// TwinCAT 3 PLC project Untitled1
// ProgramVersion: 3.1.4023.0
// libraries:
//   Tc2_MC2, * (Beckhoff Automation GmbH)
//   Tc2_Standard, * (Beckhoff Automation GmbH)
//   Tc2_System, * (Beckhoff Automation GmbH)
//   Tc3_Module, * (Beckhoff Automation GmbH)
// project tree:
//   DUTs/ stAxisIN.TcDUT, stAxisInterface.TcDUT, stAxisOut.TcDUT
//   GVLs/ GVL_Axis.TcGVL
//   / PlcTask.TcTTO
//   POUs/ FB_Motion.TcPOU, MAIN.TcPOU
// real-time tasks:
//   TASK PlcTask: cycle T#10ms, priority 20, ADS port 350
// motion (NC):
//   TASK NC-Task 1 SAF: cycle T#2ms, priority 4, ADS port 501
//   TASK NC-Task 1 SVB: cycle T#10ms, priority 8, ADS port 511
//   AXIS Axis 1 (id 1)
//     OtherSettings: AllowMotionCmdToSlave=true
//     encoder EncType=1
//     drive DrvType=5
//       Analog: TorqueSetpointScale=10, ScaleFactorActTorque=0.1
//       TimeComp: TaskDelayCycles=1
//     controller CtrType=1
//       CtrPara: PriorControlFactor=1
//         Observer: BandWidth=20
// variable links:
//   Untitled1/Untitled1 Instance <-> NC-Task 1 SAF/Axes/Axis 1
//     PlcTask Inputs/GVL_Axis.Axis1.NcToPlc <-> Outputs/ToPlc
//     PlcTask Outputs/GVL_Axis.Axis1.PlcToNc <-> Inputs/FromPlc

CONFIGURATION Untitled1
    RESOURCE PLC ON TwinCAT3
        TASK PlcTask(INTERVAL := T#10ms, PRIORITY := 20);
        PROGRAM MAIN WITH PlcTask : MAIN;
    END_RESOURCE
END_CONFIGURATION

// ---- DUTs/stAxisIN.TcDUT
TYPE stAxisIN :
STRUCT

bPower	 :	BOOL;
bStop	:	BOOL;
bMoveAbs	:	BOOL;
bReset	:	bOOL;

fOverride	:	LREAL;
fPosition	:	LREAL;
fVelocity	:	LREAL;


END_STRUCT
END_TYPE

// ---- DUTs/stAxisInterface.TcDUT
TYPE stAxisInterface :
STRUCT
	

IN	:	stAxisIN;
OUT	:	stAxisOUT;


END_STRUCT
END_TYPE

// ---- DUTs/stAxisOut.TcDUT
TYPE stAxisOut :
STRUCT
	
bPowerErr	:	BOOL;
bPowerEnabled	:	BOOL;
bPowerACTIVE	:	BOOL;

bStopDone	:	BOOL;
bStopActive	:	BOOL;
bStopErr	:	BOOL;

bMoveAbsDone	:	BOOL;
bMoveAbsBusy	:	BOOL;
bMoveAbsActive	:	BOOL;
bMoveAbsErr		:	BOOL;

bResetDone	:	BOOL;
bResetErr	:	BOOL;	

END_STRUCT
END_TYPE

// ---- GVLs/GVL_Axis.TcGVL
VAR_GLOBAL
	
Axis1 : AXIS_REF;
stAxis1	:	stAxisInterface;


END_VAR

// ---- POUs/MAIN.TcPOU
PROGRAM MAIN
VAR
	nState: INT;
	bButton	:	BOOL;
	fbMotion	:	FB_Motion;
	T1: TON;
END_VAR



stAxis1.IN.bPower	:=	TRUE;
stAxis1.IN.fOverride	:=	100;

fbMotion(Axis:=Axis1 , staxisinterface:=stAxis1 );
ACT_Motion();

ACTION ACT_Motion:
CASE nState OF 
	

	0:
	
		IF bButton AND NOT stAxis1.OUT.bPowerErr
		AND stAxis1.OUT.bPowerEnabled
		AND NOT stAxis1.OUT.bPowerErr 
		AND	NOT stAxis1.OUT.bStopActive THEN
		
			nState := 10;
		
		END_IF
		
		
	10:
	
	stAxis1.IN.bMoveAbs	:=	TRUE;
	stAxis1.IN.bStop	:=	FALSE;	
	
	stAxis1.IN.fPosition	:=	1000;
	stAxis1.IN.fVelocity	:=	500;
	
	IF stAxis1.OUT.bMoveAbsBusy 
	AND NOT stAxis1.OUT.bMoveAbsErr
	AND NOT	stAxis1.OUT.bMoveAbsErr	THEN	
	
		nState := 20;	
	
	ELSIF stAxis1.OUT.bMoveAbsErr THEN
		
		nState:=999;
		
	END_IF
	
	
	20:
	
	IF  stAxis1.OUT.bMoveAbsDone 
	AND NOT stAxis1.OUT.bMoveAbsErr THEN

		stAxis1.IN.bMoveAbs:=FALSE;
		nState:=25;	
		
		
	ELSIF stAxis1.OUT.bMoveAbsErr THEN
		
		nState := 999;
	
	END_IF
	
	
	25:
	
	T1(IN:=TRUE , PT:=T#5S, Q=> , ET=> );
	
	IF T1.Q THEN
		nState := 30;
	T1(IN:=TRUE);
	END_IF

	30:
	
	stAxis1.IN.bMoveAbs	:=	TRUE;
	stAxis1.IN.bStop	:=	FALSE;	
	
	stAxis1.IN.fPosition	:=	5000;
	stAxis1.IN.fVelocity	:=	750;
	
	IF stAxis1.OUT.bMoveAbsBusy 
	AND NOT stAxis1.OUT.bMoveAbsErr
	AND NOT	stAxis1.OUT.bMoveAbsErr	THEN	
	
		nState := 40;	
	
	ELSIF stAxis1.OUT.bMoveAbsErr THEN
		
		nState:=999;
		
	END_IF
	
	
	40:
	
	IF  stAxis1.OUT.bMoveAbsDone 
	AND NOT stAxis1.OUT.bMoveAbsErr THEN

		stAxis1.IN.bMoveAbs:=FALSE;
		nState	:=	50;	
		
		
	ELSIF stAxis1.OUT.bMoveAbsErr THEN
		
		nState := 999;
	
	END_IF
	
	
	50:
	
	stAxis1.IN.bMoveAbs	:=	TRUE;
	stAxis1.IN.bStop	:=	FALSE;	
	
	stAxis1.IN.fPosition	:=	0;
	stAxis1.IN.fVelocity	:=	1000;
	
	IF stAxis1.OUT.bMoveAbsBusy 
	AND NOT stAxis1.OUT.bMoveAbsErr
	AND NOT	stAxis1.OUT.bMoveAbsErr	THEN	
	
		nState := 60;	
	
	ELSIF stAxis1.OUT.bMoveAbsErr THEN
		
		nState:=999;
		
	END_IF
	
	
	60:
	
	IF  stAxis1.OUT.bMoveAbsDone 
	AND NOT stAxis1.OUT.bMoveAbsErr THEN

		stAxis1.IN.bMoveAbs:=FALSE;
		nState	:=	0;	
		
		
	ELSIF stAxis1.OUT.bMoveAbsErr THEN
		
		nState := 999;
	
	END_IF
	
	
	
	
END_CASE
END_ACTION

END_PROGRAM

// ---- POUs/FB_Motion.TcPOU
FUNCTION_BLOCK Fb_Motion
VAR_INPUT
END_VAR
VAR_OUTPUT
END_VAR
VAR
	
	MCPower: MC_Power;
	McStop: MC_Stop;
	MCMoveAbs: MC_MoveAbsolute;
	McReset: MC_Reset;
	
END_VAR
VAR_IN_OUT
	
	Axis : AXIS_REF;
	staxisinterface : stAxisInterface;

END_VAR

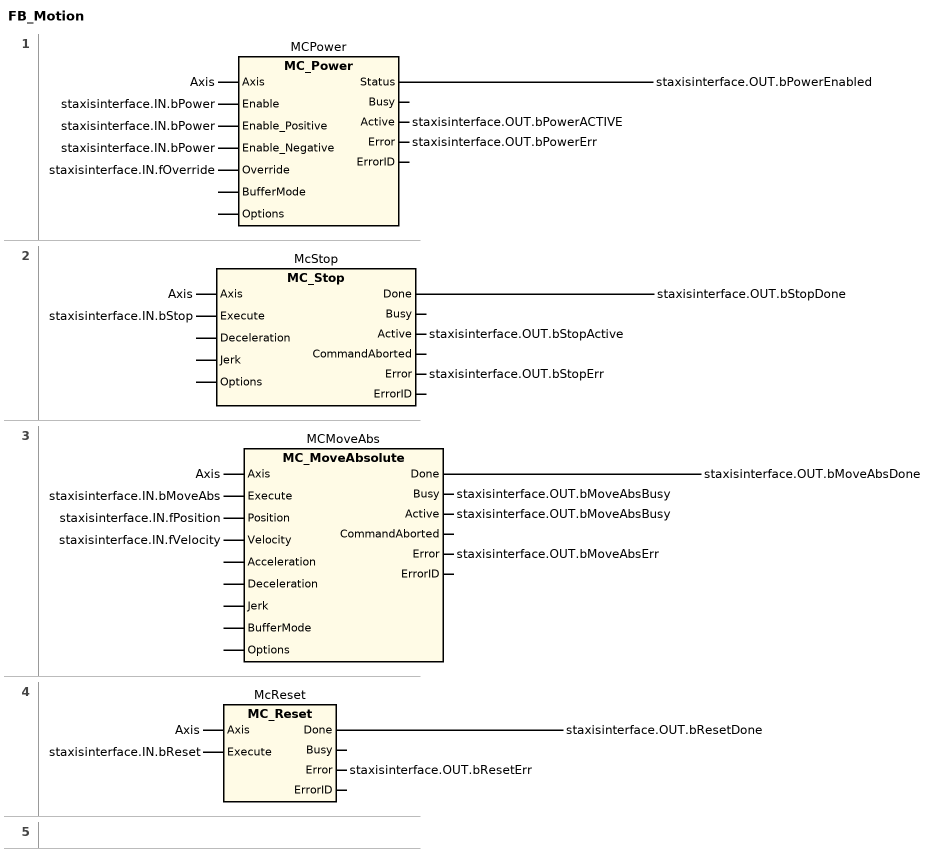
// NETWORK 1
MCPower(
    Axis := Axis,
    Enable := staxisinterface.IN.bPower,
    Enable_Positive := staxisinterface.IN.bPower,
    Enable_Negative := staxisinterface.IN.bPower,
    Override := staxisinterface.IN.fOverride,
    Active => staxisinterface.OUT.bPowerACTIVE,
    Error => staxisinterface.OUT.bPowerErr); // MC_Power
staxisinterface.OUT.bPowerEnabled := MCPower.Status;

// NETWORK 2
McStop(
    Axis := Axis,
    Execute := staxisinterface.IN.bStop,
    Active => staxisinterface.OUT.bStopActive,
    Error => staxisinterface.OUT.bStopErr); // MC_Stop
staxisinterface.OUT.bStopDone := McStop.Done;

// NETWORK 3
MCMoveAbs(
    Axis := Axis,
    Execute := staxisinterface.IN.bMoveAbs,
    Position := staxisinterface.IN.fPosition,
    Velocity := staxisinterface.IN.fVelocity,
    Busy => staxisinterface.OUT.bMoveAbsBusy,
    Active => staxisinterface.OUT.bMoveAbsBusy,
    Error => staxisinterface.OUT.bMoveAbsErr); // MC_MoveAbsolute
staxisinterface.OUT.bMoveAbsDone := MCMoveAbs.Done;

// NETWORK 4
McReset(Axis := Axis, Execute := staxisinterface.IN.bReset, Error => staxisinterface.OUT.bResetErr); // MC_Reset
staxisinterface.OUT.bResetDone := McReset.Done;

// NETWORK 5

END_FUNCTION_BLOCK
